Staubli VAL3: ReplyType.dtx

public num nSuccess = 1
public num nFailure = 2
